(* CODESYS project LD_PROGRAMM.pou_xml.xml

Project tree, tasks and I/O mapping:
  program LD_PROGRAMM [LD]
*)

// LD_PROGRAMM
PROGRAM LD_PROGRAMM
VAR
	xStart : BOOL;
	xStop_NC : BOOL;
	xPump : BOOL;
	xLamp : BOOL;
	
	timer : TON;
	
	LD_FB_Instance : LD_FB;
END_VAR

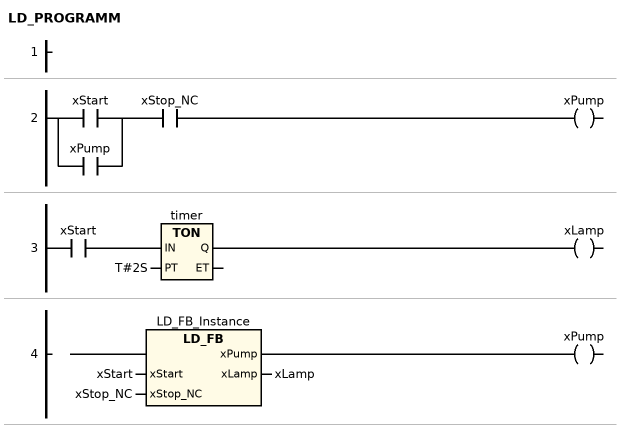
// NETWORK 1

// NETWORK 2
xPump := (xStart OR xPump) AND xStop_NC;

// NETWORK 3
timer(IN := xStart, PT := T#2S); // TON
xLamp := timer.Q;

// NETWORK 4
LD_FB_Instance(xStart := xStart, xStop_NC := xStop_NC, xLamp => xLamp); // LD_FB
xPump := LD_FB_Instance.xPump;

END_PROGRAM
